# EPICS substitutions: elioApp/Db/EL3318.substitutions
file EL331x.template { pattern
{ CHAN	}
{ 1	}
{ 2	}
{ 3	}
{ 4	}
{ 5	}
{ 6	}
{ 7	}
{ 8	}
}
